{attribute 'Tc2GvlVarNames'}
{attribute 'strict'}
//Riferimento origine assi postazione in WA rispetto l'origine degli assi
TYPE e_OrdinamentoPostazione :
(
	NOT_DEFINED		:= -1,
	CRESCENTE	 	:= 1,	(* Identifica che LA numerazione CRESCE dall'origine della macchina *)
	DECRESCENTE	 	:= 2	(* Identifica che LA numerazione DECRESCE dall'origine della macchina *)	
);
END_TYPE
//  NOT_DEFINED = '-1'

(* stored: Version 1.1.0.1, ProductVersion 3.1.4024.9
   EnumerationTextList e_OrdinamentoPostazione: Id {ab6a40f6-afcb-4605-a738-4f7b980f15d1} *)
